TYPE ST_Candle :
STRUCT
	dia			: REAL;
	height 		: REAL;
	numWicks 	: INT;
	weight 		: REAL;
END_STRUCT
END_TYPE

(* stored: Version 1.1.0.1, ProductVersion 3.1.4024.12
   DUT ST_Candle: Id {e7e915a0-ba52-49f3-bd14-5126f3ee3ad9} *)
